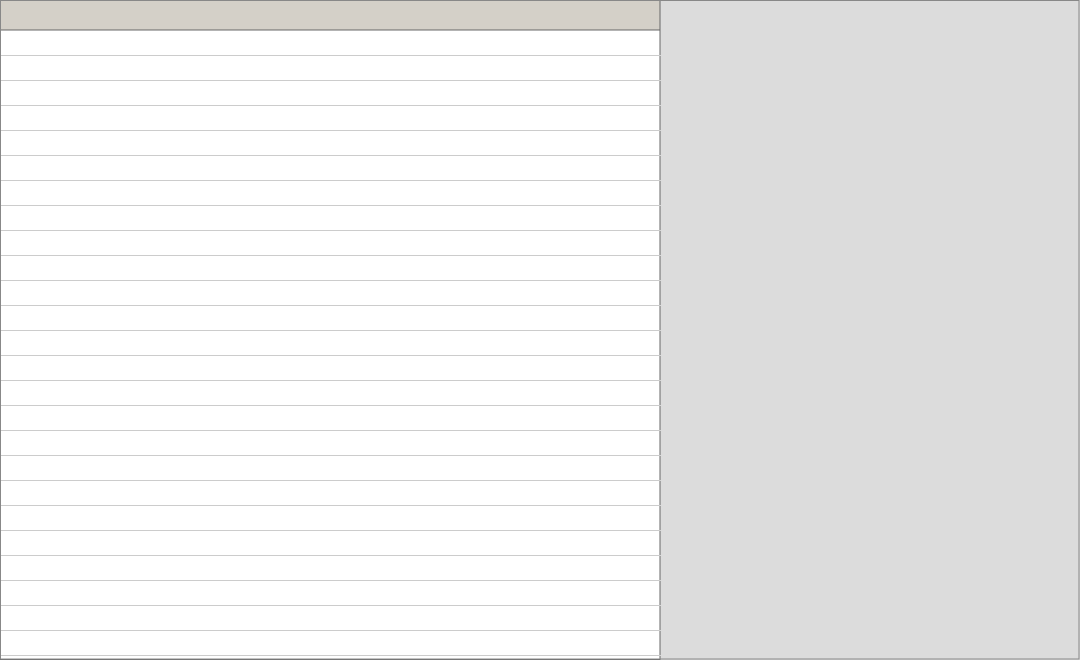
VISUALIZATION Page_Alarms  // 1080x660, background image 
    Table (0,0 660x660), data array: GVL_Modules.g_unMachine.s_stHmi.fbHmiAlarmCollector.s_stHmi.asAlarmList
        p3854506369: GVL_Modules.g_unMachine.s_stHmi.fbHmiAlarmCollector.s_stHmi.asAlarmList[INDEX]
        p1014161805: Param_Alarms.c_nMaxNrOfListEntries - 1 + INT#1
END_VISUALIZATION

(* stored: Version 1.1.0.1, ProductVersion 3.1.4026.13
   Visu Page_Alarms: Id {721454e9-b26f-43ff-9b12-a8903a2cbf43} *)
